FUNCTION_BLOCK FB_PVPROG_00 (* Composite Function Block that implements the PVprog algorithm *)
  (* Standard: 61499-2; Description: IEC 61499 implementation of the "PVprog" algorithm. Original version's MIT license: Copyright (c) 2016 Joseph Bergner, Johannes Weniger, Tjarko Tjaden Permission is hereby granted, free of charge, to any person obtaining a copy of this software and associated documentation files (the "Software"), to deal in the Software without restriction, including without limitation the rights to use, copy, modify, merge, publish, distribute, sublicense, and/or sell copies of the Software, and to permit persons to whom the Software is furnished to do so, subject to the following conditions: The above copyright notice and this permission notice shall be included in all copies or substantial portions of the Software. THE SOFTWARE IS PROVIDED "AS IS", WITHOUT WARRANTY OF ANY KIND, EXPRESS OR IMPLIED, INCLUDING BUT NOT LIMITED TO THE WARRANTIES OF MERCHANTABILITY, FITNESS FOR A PARTICULAR PURPOSE AND NONINFRINGEMENT. IN NO EVENT SHALL THE AUTHORS OR COPYRIGHT HOLDERS BE LIABLE FOR ANY CLAIM, DAMAGES OR OTHER LIABILITY, WHETHER IN AN ACTION OF CONTRACT, TORT OR OTHERWISE, ARISING FROM, OUT OF OR IN CONNECTION WITH THE SOFTWARE OR THE USE OR OTHER DEALINGS IN THE SOFTWARE. *)
  (* Version 1.0, 2017-05-22, Marc Jakobi, HTW Berlin *)
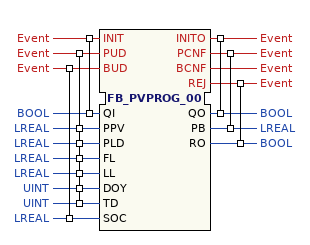
  EVENT_INPUT
    INIT WITH QI; (* Initialization Request *)
    PUD WITH PPV, PLD, FL, LL, DOY, TD; (* Power Update Event *)
    BUD WITH SOC; (* Battery Update Event *)
  END_EVENT
  EVENT_OUTPUT
    INITO WITH QO; (* Initialization Confirm *)
    PCNF WITH PB; (* Power Update Confirmation *)
    BCNF; (* Battery Update Confirmation *)
    REJ WITH RO; (* Request Rejection Notification *)
  END_EVENT
  VAR_INPUT
    QI : BOOL; (* Input event qualifier *)
    PPV : LREAL; (* PV power in W *)
    PLD : LREAL; (* Load in W *)
    FL : LREAL; (* Feed-in limitation in W (0 for none) *)
    LL : LREAL; (* Load limit in W (0 for none) *)
    DOY : UINT := 1; (* Day of the year [1..365] *)
    TD : UINT; (* Time of day [min] [0..1439] *)
    SOC : LREAL := 0.2; (* State of charge of the battery [0..1] *)
  END_VAR
  VAR_OUTPUT
    QO : BOOL; (* Output event qualifier *)
    PB : LREAL; (* Set battery charging power in W (positive = charge, negative = discharge) *)
    RO : BOOL; (* Rejection reason indicator. TRUE: Not enough time passed; FALSE: Currently locked *)
  END_VAR
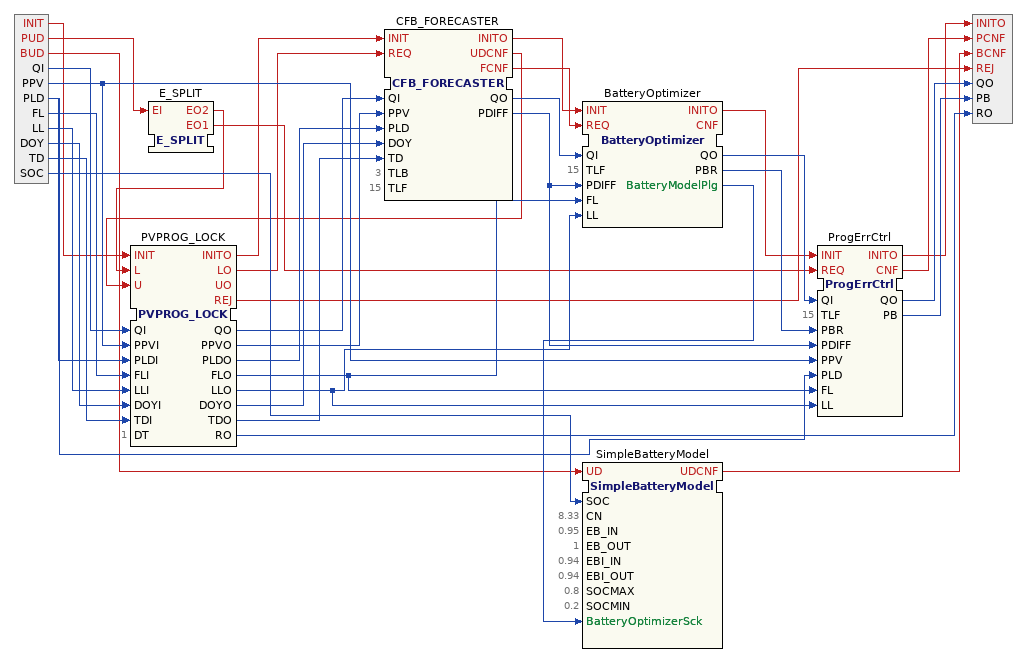
  FBS
    CFB_FORECASTER : CFB_FORECASTER(TLB := 3, TLF := 15);
    PVPROG_LOCK : PVPROG_LOCK(DT := 1);
    ProgErrCtrl : ProgErrCtrl(TLF := 15);
    BatteryOptimizer : BatteryOptimizer(TLF := 15);
    SimpleBatteryModel : SimpleBatteryModel(CN := 8.33, EB_IN := 0.95, EB_OUT := 1, EBI_IN := 0.94, EBI_OUT := 0.94, SOCMAX := 0.8, SOCMIN := 0.2);
    E_SPLIT : E_SPLIT;
  END_FBS
  EVENT_CONNECTIONS
    INIT TO PVPROG_LOCK.INIT;
    PVPROG_LOCK.INITO TO CFB_FORECASTER.INIT;
    PVPROG_LOCK.REJ TO REJ;
    PVPROG_LOCK.LO TO CFB_FORECASTER.REQ;
    ProgErrCtrl.INITO TO INITO;
    CFB_FORECASTER.INITO TO BatteryOptimizer.INIT;
    CFB_FORECASTER.FCNF TO BatteryOptimizer.REQ;
    BatteryOptimizer.INITO TO ProgErrCtrl.INIT;
    BUD TO SimpleBatteryModel.UD;
    SimpleBatteryModel.UDCNF TO BCNF;
    PUD TO E_SPLIT.EI;
    E_SPLIT.EO2 TO PVPROG_LOCK.L;
    E_SPLIT.EO1 TO ProgErrCtrl.REQ;
    CFB_FORECASTER.UDCNF TO PVPROG_LOCK.U;
    ProgErrCtrl.CNF TO PCNF;
  END_CONNECTIONS
  DATA_CONNECTIONS
    QI TO PVPROG_LOCK.QI;
    PPV TO PVPROG_LOCK.PPVI;
    PLD TO PVPROG_LOCK.PLDI;
    FL TO PVPROG_LOCK.FLI;
    LL TO PVPROG_LOCK.LLI;
    DOY TO PVPROG_LOCK.DOYI;
    TD TO PVPROG_LOCK.TDI;
    PVPROG_LOCK.QO TO CFB_FORECASTER.QI;
    PVPROG_LOCK.DOYO TO CFB_FORECASTER.DOY;
    PVPROG_LOCK.TDO TO CFB_FORECASTER.TD;
    PVPROG_LOCK.RO TO RO;
    PVPROG_LOCK.PPVO TO CFB_FORECASTER.PPV;
    PVPROG_LOCK.PLDO TO CFB_FORECASTER.PLD;
    CFB_FORECASTER.PDIFF TO ProgErrCtrl.PDIFF;
    PVPROG_LOCK.FLO TO ProgErrCtrl.FL;
    PVPROG_LOCK.LLO TO ProgErrCtrl.LL;
    ProgErrCtrl.QO TO QO;
    ProgErrCtrl.PB TO PB;
    CFB_FORECASTER.QO TO BatteryOptimizer.QI;
    CFB_FORECASTER.PDIFF TO BatteryOptimizer.PDIFF;
    PVPROG_LOCK.FLO TO BatteryOptimizer.FL;
    PVPROG_LOCK.LLO TO BatteryOptimizer.LL;
    BatteryOptimizer.QO TO ProgErrCtrl.QI;
    BatteryOptimizer.PBR TO ProgErrCtrl.PBR;
    SOC TO SimpleBatteryModel.SOC;
    BatteryOptimizer.BatteryModelPlg TO SimpleBatteryModel.BatteryOptimizerSck;
    PPV TO ProgErrCtrl.PPV;
    PLD TO ProgErrCtrl.PLD;
  END_CONNECTIONS
END_FUNCTION_BLOCK
